TYPE EtcSlaveBase_82538BE2 :
STRUCT
END_STRUCT
END_TYPE

(* stored: Version 1.2.0.0, ProductVersion 3.1.4024.11
   DUT EtcSlaveBase_82538BE2: Id {ea046009-6cf5-4226-a6b1-d3ce8fdcf781} *)
